{attribute 'strict'}
//Pathing Enum
TYPE E_CompressionStages :
(
	Bypass_Line:=1,
    Second_Stage_Compression:=2,
    First_Stage_Compression:=3
)USINT;
END_TYPE

(* stored: Version 1.1.0.1
   DUT E_CompressionStages: Id {6b108da2-1011-4f56-a624-371ad8ec33b9} *)
